// Mitsubishi GX Works2 project: bmov   PLC: Q02/Q02H

PROGRAM MAIN
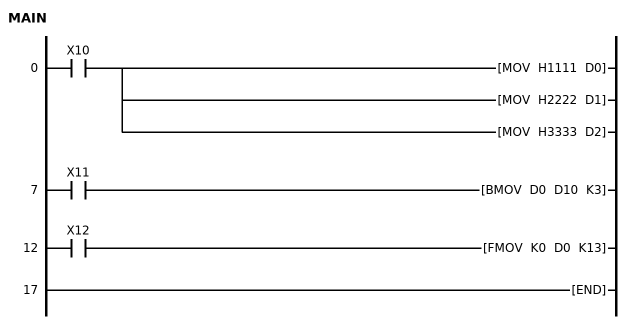
0     LD      X10
      MOV     H1111 D0
      MOV     H2222 D1
      MOV     H3333 D2
7     LD      X11
      BMOV    D0 D10 K3
12    LD      X12
      FMOV    K0 D0 K13
17    END
END_PROGRAM
